// TIA Portal project "Ejemplo_2" (V16)

(* hardware
DEVICE "S7300/ET200M station_1"  S7-300 station
   slot 0: "Perfil soporte_0"  Rail  6ES7 390-1***0-0AA0
   slot 2: "PLC_1"  CPU 313C  6ES7 313-5BG04-0AB0  V3.3
      slot 0: "Interfaz MPI_1"  MPI
      slot 2: "DI 24/DO 16_1"  DI24/DO16
      slot 3: "AI 5/AO 2_1"  AI5/AO2
      slot 4: "Contaje_1"  Counter
*)

// ===== PLC "PLC_1"  CPU 313C =====

VAR_GLOBAL   // PLC tag table "Tabla de variables estándar"
   "Contador" AT %MD0 : DInt;
   "Tag_1" AT %M0.0 : Bool;
END_VAR

ORGANIZATION_BLOCK "Main"   // OB1, LAD
TITLE = "Main Program Sweep (Cycle)"
{ S7_Optimized_Access := 'FALSE' }
VERSION : 0.1
   VAR_TEMP
      OB1_EV_CLASS : Byte;   // Bits 0-3 = 1 (Coming event), Bits 4-7 = 1 (Event class 1)
      OB1_SCAN_1 : Byte;   // 1 (Cold restart scan 1 of OB 1), 3 (Scan 2-n of OB 1)
      OB1_PRIORITY : Byte;   // Priority of OB Execution
      OB1_OB_NUMBR : Byte;   // 1 (Organization block 1, OB1)
      OB1_RESERVED_1 : Byte;   // Reserved for system
      OB1_RESERVED_2 : Byte;   // Reserved for system
      OB1_PREV_CYCLE : Int;   // Cycle time of previous OB1 scan (milliseconds)
      OB1_MIN_CYCLE : Int;   // Minimum cycle time of OB1 (milliseconds)
      OB1_MAX_CYCLE : Int;   // Maximum cycle time of OB1 (milliseconds)
      OB1_DATE_TIME : Date_And_Time;   // Date and time OB1 started
   END_VAR
BEGIN
END_ORGANIZATION_BLOCK

ORGANIZATION_BLOCK "HW_INT0"   // OB40, LAD
TITLE = "Hardware Interrupt"
{ S7_Optimized_Access := 'FALSE' }
VERSION : 0.1
   VAR_TEMP
      OB40_EV_CLASS : Byte;   // Bits 0-3 = 1 (Coming event), Bits 4-7 = 1 (Event class 1)
      OB40_STRT_INF : Byte;   // 16#41 (OB 40 has started)
      OB40_PRIORITY : Byte;   // Priority of OB Execution
      OB40_OB_NUMBR : Byte;   // 40 (Organization block 40, OB40)
      OB40_RESERVED_1 : Byte;   // Reserved for system
      OB40_IO_FLAG : Byte;   // 16#54 (input module), 16#55 (output module)
      OB40_MDL_ADDR : Word;   // Base address of module initiating interrupt
      OB40_POINT_ADDR : DWord;   // Interrupt status of the module
      OB40_DATE_TIME : Date_And_Time;   // Date and time OB40 started
   END_VAR
BEGIN

REGION Network 1
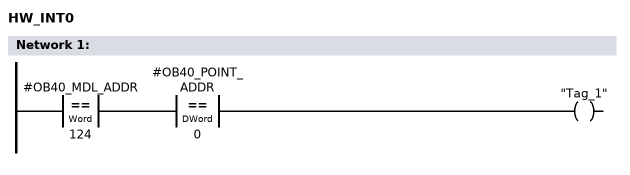
   RUNG wire#powerrail
      { S7_Templates := "SrcType := Word" } EQ_Contact(in1 := #OB40_MDL_ADDR, in2 := 124)
      { S7_Templates := "SrcType := DWord" } EQ_Contact(in1 := #OB40_POINT_ADDR, in2 := 0)
      Coil( "Tag_1" )
   END_RUNG
   // the same network as SCL:
   "Tag_1" := (#OB40_MDL_ADDR = 124) AND (#OB40_POINT_ADDR = 0);
END_REGION
END_ORGANIZATION_BLOCK